FUNCTION_BLOCK operate (* Basic Function Block Type *)
  (* Standard: 61499-2 *)
  (* Version 0.0, 24/03/2016, Chen-Wei, nxtControl GmbH, Template *)
  PACKAGE Main;
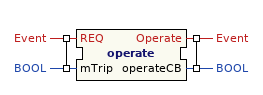
  EVENT_INPUT
    REQ WITH mTrip; (* Normal Execution Request *)
  END_EVENT
  EVENT_OUTPUT
    Operate WITH operateCB; (* Execution Confirmation *)
  END_EVENT
  VAR_INPUT
    mTrip : BOOL;
  END_VAR
  VAR_OUTPUT
    operateCB : BOOL; (* Output event qualifier *)
  END_VAR
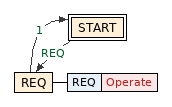
  EC_STATES
    START; (* Initial State *)
    REQ : REQ -> Operate; (* Normal execution *)
  END_STATES
  EC_TRANSITIONS
    START TO REQ := REQ;
    REQ TO START := 1;
  END_TRANSITIONS
  ALGORITHM REQ IN ST: (* Normally executed algorithm *)
REQ := 0;
operateCB := mTrip;

;
  END_ALGORITHM
END_FUNCTION_BLOCK
